% RSLogix 500 project P1.RSS, saved by version 8.30.00.16 %
PROJECT "UNTITLED"    % processor: Bul.1763 MicroLogix 1100 Series B %

PROGRAM FILES
  LAD 2   3 rungs
  LAD 3 "IO"  5 rungs
  LAD 4 "CTRL"  7 rungs

DATA FILES
  O0 OUTPUT  4 elements
  I1 INPUT  6 elements
  S2 STATUS  66 elements
  B3 BINARY  1 elements
  T4 TIMER  1 elements
  C5 COUNTER  1 elements
  R6 CONTROL  1 elements
  N7 INTEGER  1 elements
  F8 FLOAT  1 elements

LADDER 2
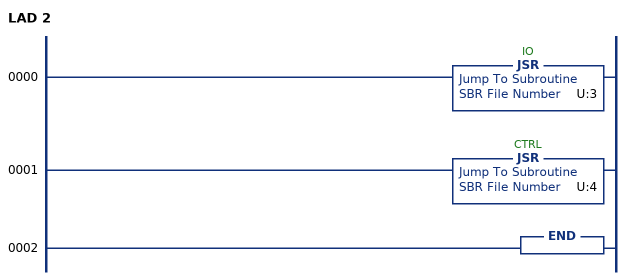
% Rung: 0 %
SOR JSR U:3 EOR
%   U:3  "IO" %
% Rung: 1 %
SOR JSR U:4 EOR
%   U:4  "CTRL" %
% Rung: 2 %
SOR END EOR

LADDER 3 "IO"
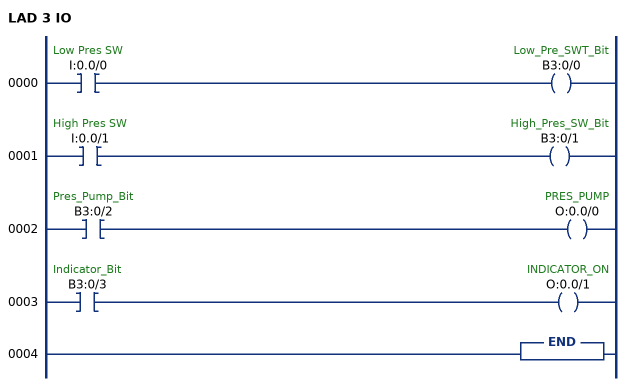
% Rung: 0 %
SOR XIC I:0.0/0 OTE B3:0/0 EOR
%   I:0.0/0  "Low Pres SW" %
%   B3:0/0  "Low_Pre_SWT_Bit" %
% Rung: 1 %
SOR XIC I:0.0/1 OTE B3:0/1 EOR
%   I:0.0/1  "High Pres SW" %
%   B3:0/1  "High_Pres_SW_Bit" %
% Rung: 2 %
SOR XIC B3:0/2 OTE O:0.0/0 EOR
%   B3:0/2  "Pres_Pump_Bit" %
%   O:0.0/0  "PRES_PUMP" %
% Rung: 3 %
SOR XIC B3:0/3 OTE O:0.0/1 EOR
%   B3:0/3  "Indicator_Bit" %
%   O:0.0/1  "INDICATOR_ON" %
% Rung: 4 %
SOR END EOR

LADDER 4 "CTRL"
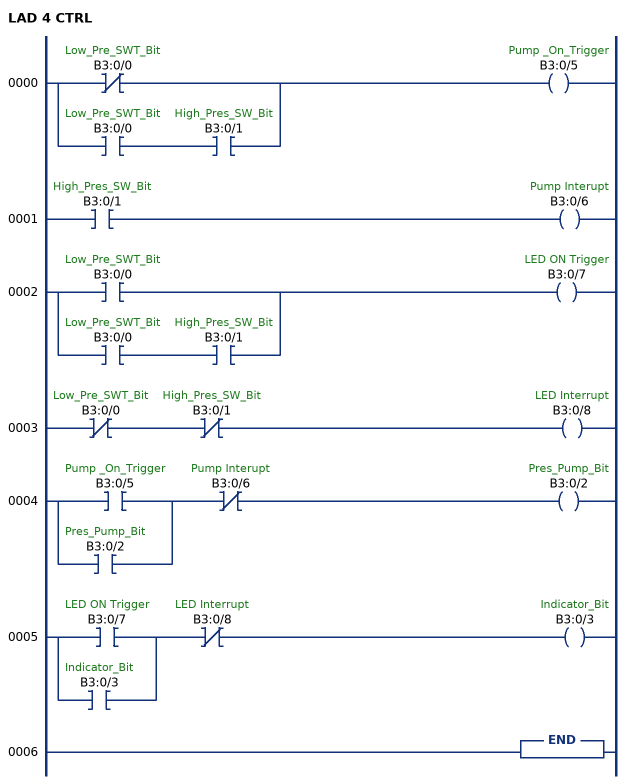
% Rung: 0 %
SOR BST XIO B3:0/0 NXB XIC B3:0/0 XIC B3:0/1 BND OTE B3:0/5 EOR
%   B3:0/0  "Low_Pre_SWT_Bit" %
%   B3:0/1  "High_Pres_SW_Bit" %
%   B3:0/5  "Pump _On_Trigger" %
% Rung: 1 %
SOR XIC B3:0/1 OTE B3:0/6 EOR
%   B3:0/1  "High_Pres_SW_Bit" %
%   B3:0/6  "Pump Interupt" %
% Rung: 2 %
SOR BST XIC B3:0/0 NXB XIC B3:0/0 XIC B3:0/1 BND OTE B3:0/7 EOR
%   B3:0/0  "Low_Pre_SWT_Bit" %
%   B3:0/1  "High_Pres_SW_Bit" %
%   B3:0/7  "LED ON Trigger" %
% Rung: 3 %
SOR XIO B3:0/0 XIO B3:0/1 OTE B3:0/8 EOR
%   B3:0/0  "Low_Pre_SWT_Bit" %
%   B3:0/1  "High_Pres_SW_Bit" %
%   B3:0/8  "LED Interrupt" %
% Rung: 4 %
SOR BST XIC B3:0/5 NXB XIC B3:0/2 BND XIO B3:0/6 OTE B3:0/2 EOR
%   B3:0/5  "Pump _On_Trigger" %
%   B3:0/2  "Pres_Pump_Bit" %
%   B3:0/6  "Pump Interupt" %
% Rung: 5 %
SOR BST XIC B3:0/7 NXB XIC B3:0/3 BND XIO B3:0/8 OTE B3:0/3 EOR
%   B3:0/7  "LED ON Trigger" %
%   B3:0/3  "Indicator_Bit" %
%   B3:0/8  "LED Interrupt" %
% Rung: 6 %
SOR END EOR
